ABB RobotStudio station: Autoclasiffier_Vacuostato_20181218-112255.rsstn

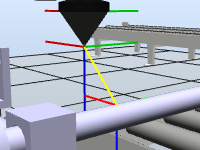
Station Station (saved by RobotStudio 6.6.7701.1025)
Controller Sistema12, task T_ROB1: task frame (RAPID world) sits at (920, -1100, 0) mm, rotated rx 0 ry 0 rz 180 deg in the station
Controller Sistema10, task T_ROB1: task frame (RAPID world) sits at (-920, -900, 0) mm in the station
Controller Sistema10
  mechanical unit ROB_1: JUAN, 6 joints, base frame (0, 0, 0) mm
Controller Sistema12
  mechanical unit ROB_1: ROBERTO, 6 joints, base frame (0, 0, 0) mm
Layout (positions relative to the parent item):
  - JUAN [mechanism, from Robots\IRB1600_6_145_G_02.rslib] at (-920, -900, 0) mm; joint values [-0.0666, 0.152, 0.4153, 3.1416, -1.0035, -0.0666] (rad or m)
  - ROBERTO [mechanism, from Robots\IRB1600_6_145_G_02.rslib] at (920, -1100, 0) mm, rotated rx 0 ry 0 rz 180 deg; joint values [-0.4677, 0.0079, -0.0561, 0.0825, 1.1142, -0.2191] (rad or m)
  - 600_guide [part, from Equipment\Conveyor Guide 600.rslib] at (3800, 50, 0) mm, rotated rx 0 ry 0 rz 180 deg
  - 4800_3str_h2 [part, from Equipment\Conveyor 4800 3str h2.rslib] at (0, -5364.61, 0) mm
  - 950_4800_h2 [part, from Equipment\Conveyor 950 4800 h2.rslib] at (475, -3400, 0) mm, rotated rx 0 ry 0 rz 90 deg
  - Pieza_5 [part] at (920, -500, 775) mm
  - Componente inteligente_1 [smart component]
      signals: DI dedo_Juan, DO Aspira
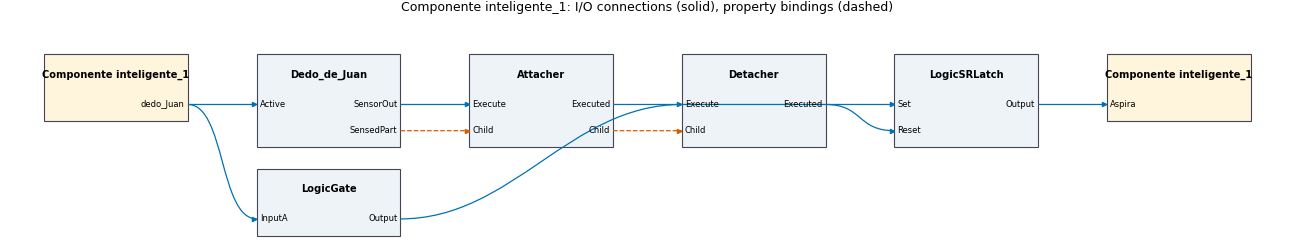
      connections:
        Dedo_de_Juan.SensorOut -> Attacher.Execute
        LogicGate.Output -> Detacher.Execute
        Componente inteligente_1.dedo_Juan -> Dedo_de_Juan.Active
        Componente inteligente_1.dedo_Juan -> LogicGate.InputA
        Attacher.Executed -> LogicSRLatch.Set
        LogicSRLatch.Output -> Componente inteligente_1.Aspira
        Detacher.Executed -> LogicSRLatch.Reset
        Dedo_de_Juan.SensedPart => Attacher.Child
        Attacher.Child => Detacher.Child
    - Dedo_de_Roberto [smart component, from Components\LineSensor.rslib] at (215.98, -749.84, 1158.66) mm, rotated rx 178.39 ry -29.24 rz 165.19 deg
        properties: Start=[0 0 0]; End=[0 0 0.035]; Radius=0.002; SensedPart=Pieza_7; SensedPoint=[0.215981719970703 -0.749844604492187 1.15866088867188]
      - _sensorPart_ [part]
    - Attacher [smart component, from Components\Attacher.rslib]
        properties: Parent=Mano_de_Juan; Flange=0; Child=(none); Mount=false; Offset=[0 0 0]; Orientation=[0 0 0]
    - LogicGate [smart component, from Components\LogicGate.rslib] at (-1050.67, 0, 0) mm
        properties: Operator=NOT; Delay=0
    - Dedo_de_Juan [smart component, from Components\LineSensor.rslib] at (-159.7, -950.69, 788.04) mm, rotated rx 180 ry 0 rz 0 deg
        properties: Start=[0 0 0]; End=[0 0 0.035]; Radius=0.002; SensedPart=(none); SensedPoint=[0 0 0]
      - _sensorPart_ [part]
    - Detacher [smart component, from Components\Detacher.rslib]
        properties: Child=(none); KeepPosition=true
    - LogicSRLatch [smart component, from Components\LogicSRLatch.rslib]
  - Mano_de_Roberto [mechanism] at (215.98, -749.84, 1158.66) mm, rotated rx -1.61 ry -29.24 rz 165.19 deg
      links: Pieza_7
  - Mano_de_Juan [mechanism] at (-159.7, -950.69, 791.04) mm, rotated rx 0 ry 0 rz 180 deg
      links: Pieza_7
  - chasis_t [part] at (-230, -1000, 595) mm, rotated rx 180 ry 0 rz 90 deg
  - Pieza_6 [part] at (370, -1250, 415) mm, rotated rx 0 ry -90 rz 0 deg
  - Componente inteligente_2 [smart component]
Attachment: Mano_de_Juan is attached to JUAN / Link6
Attachment: Dedo_de_Roberto is attached to Mano_de_Roberto / Pieza_7
Attachment: Dedo_de_Juan is attached to Mano_de_Juan / Pieza_7
Attachment: Mano_de_Roberto is attached to ROBERTO / Link6
Targets, tools, work objects and paths stored in the station, written as RAPID:
! task T_ROB1
MODULE CalibData
  PERS tooldata Ventosa1:=[TRUE,[[0.000009563,-0.000007568,35],[1,0,0,0]],[1,[0,0,1],[1,0,0,0],0,0,0]];
ENDMODULE

! task T_ROB1
MODULE Module1
  CONST robtarget Target_10:=[[710.302,-50.687,706.042],[0,1,0,0],[0,0,0,0],[9E+09,9E+09,9E+09,9E+09,9E+09,9E+09]];
  CONST robtarget Target_20:=[[760.301980587,-50.686989693,756.042035513],[-0.000000033,1,-0.000000027,0.000000018],[-1,1,-1,1],[9E+09,9E+09,9E+09,9E+09,9E+09,9E+09]];
  PROC Path_10()
    MoveL Target_10,v1000,z100,Ventosa1\WObj:=wobj0;
    MoveL Target_20,v1000,z100,Ventosa1\WObj:=wobj0;
  ENDPROC
ENDMODULE

